// TIA Portal V18 export
DATA_BLOCK "man_descrete_sr_DB"   // DB28
VERSION : 0.1
// stored: AutoNumber true, DBAccessibleFromOPCUA true, InstanceOfName man_descrete_sr, InstanceOfType FB
"man_descrete_sr"
   // VAR_INPUT
   //    condions : Bool;
   //    buttons : Bool;
   //    arrived : Bool;
   // END_VAR
   // VAR_OUTPUT
   //    exce_man : Bool;
   // END_VAR
BEGIN
END_DATA_BLOCK
